Universal Robots URScript: T014_qwen2.5-coder_32b_adversarial_A8.6_rep1.urscript

def hybrid_multi_angle_inspection():
    # Move to Home position at max joint speed
    movej(p[0, -90, 90, -180, 45, 0], a=1.2, v=1.2)

    # Move to Top-down view position
    movel(p[x_top, y_top, z_top, rx_top, ry_top, rz_top], a=1.2, v=1.2)

    # Move to Side view position
    movel(p[x_side, y_side, z_side, rx_side, ry_side, rz_side], a=1.2, v=1.05)

    # Move to Angled view position
    movel(p[x_angled, y_angled, z_angled, rx_angled, ry_angled, rz_angled], a=1.2, v=1.05)

    # Retract from inspection positions
    movel(p[x_retract, y_retract, z_retract, rx_retract, ry_retract, rz_retract], a=1.2, v=1.2)

    # Additional move (not specified in the task description)
    # Placeholder for any additional motion required
    movel(p[x_additional, y_additional, z_additional, rx_additional, ry_additional, rz_additional], a=1.2, v=1.2)

end

# Call the function to execute the inspection sequence
hybrid_multi_angle_inspection()
